// TIA Portal V19 export
// export: Created 2026-08-20T21:47:31.0593778Z, ExportSetting WithDefaults, DisplayName Totally Integrated Automation Portal, DisplayVersion V19, DisplayName TIA Portal Openness, DisplayVersion V19, DisplayName TIA Portal Version Control Interface, DisplayVersion V19, DisplayName STEP 7 Professional, DisplayVersion V19, DisplayName STEP 7 Safety, DisplayVersion V19, DisplayName WinCC Basic/Comfort/Advanced, DisplayVersion V19, DisplayName WinCC Unified, DisplayVersion V19
FUNCTION_BLOCK "FB_PumpDown"   // FB3, SCL
{ S7_Optimized_Access := 'TRUE' }
VERSION : 0.1
// Roughing pump-down sequence.
//  generated by LADDER - do not edit by hand
// stored: AutoNumber true, IsIECCheckEnabled false, IsRetainMemResEnabled false, MemoryReserve 100, SetENOAutomatically false, UDAEnableTagReadback false
   VAR
      stable_ok : Bool;   // Pressure stable timer done
      T_stable_t { S7_SetPoint := 'True'} : TON_TIME;   // instance for timer T_stable
   END_VAR
BEGIN
       // timer TON T_stable: Pressure must hold for 10 s before declaring vacuum.
       #T_stable_t(IN := "pressure_ok",
                   PT := T#10s);
       #stable_ok := #T_stable_t.Q;
       // state_machine SM_pumpdown: IDLE -> PUMPING -> AT_VACUUM, with fault fallback.
       CASE "pumpdown_state" OF
           0:  (* IDLE *)
               "pump_start_cmd" := FALSE;
               "at_vacuum" := FALSE;
               IF "pumpdown_request" THEN
                   "pumpdown_state" := 1;
               END_IF;
           1:  (* PUMPING *)
               "pump_start_cmd" := TRUE;
               IF "pump_fault_alarm" THEN
                   "pumpdown_state" := 99;
               ELSIF #stable_ok THEN
                   "pumpdown_state" := 2;
               END_IF;
           2:  (* AT_VACUUM *)
               "at_vacuum" := TRUE;
               IF NOT "pressure_ok" THEN
                   "pumpdown_state" := 1;
               ELSIF NOT "pumpdown_request" THEN
                   "pumpdown_state" := 0;
               END_IF;
           99:  (* FAULT *)
               "pump_start_cmd" := FALSE;
               "at_vacuum" := FALSE;
               IF "reset_pb" AND NOT "pump_fault_alarm" THEN
                   "pumpdown_state" := 0;
               END_IF;
       END_CASE;
END_FUNCTION_BLOCK
